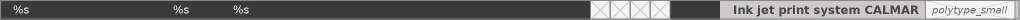
VISUALIZATION VISU_Header  // 1020x20
    Rectangle (0,0 1020x20)
    Rectangle (10,0 160x20), "%s", text variable: PRG_SYSTEM.sC_Ads_System.aProject
    Rectangle (170,0 60x20), "%s", text variable: PRG_SYSTEM.sC_Ads_System.aMachine
    Rectangle (230,0 120x20), "%s", text variable: PRG_SYSTEM.aCurrentDateTime
    Image (650,0 20x20), invisible if: NOT PRG_MACHINE.bO_ErrorMsgActive, image: GlobalImagePool.error_icon
    Image (610,0 20x20), invisible if: NOT PRG_MACHINE.sO_SystemCmd.bEStop, image: GlobalImagePool.estop_icon
    Image (590,0 20x20), invisible if: NOT PRG_MACHINE.sO_SystemCmd.bSleep, image: GlobalImagePool.sleep_icon
    Image (630,0 20x20), invisible if: NOT PRG_MACHINE.bO_WarningMsgActive, image: GlobalImagePool.warning_icon
    Rectangle (720,0 300x20)
    Image (925,0 90x20), image: polytype_small
    Rectangle (730,0 200x20), "Ink jet print system CALMAR"
END_VISUALIZATION

(* stored: Version 1.1.0.1, ProductVersion 3.1.4024.11
   Visu VISU_Header: Id {8e7baa27-1065-49fa-8d43-9a1850979f1d} *)
